// TIA Portal V17 export
// export: Created 2024-01-30T08:49:13.4989506Z, ExportSetting WithDefaults, DisplayName Totally Integrated Automation Portal, DisplayVersion V17 Update 6, DisplayName TIA Portal Openness, DisplayVersion V17 Update 6, DisplayName TIA Portal Version Control Interface, DisplayVersion V17, DisplayName STEP 7 Professional, DisplayVersion V17 Update 6, DisplayName STEP 7 Safety, DisplayVersion V17 Update 6, DisplayName WinCC Advanced, DisplayVersion V17 Update 6
FUNCTION "AnalogMeasurement" : Void   // FC2, LAD
{ S7_Optimized_Access := 'TRUE' }
VERSION : 0.1
// stored: AutoNumber true, IsIECCheckEnabled false, SetENOAutomatically false, UDAEnableTagReadback false
   VAR_INPUT
      "LK-H057_01" : Int;   // Keyence Dist.Senz-01
      "LK-H057_02" : Int;   // Keyence Dist.Senz-01
   END_VAR
   VAR_OUTPUT
      "LK-H057_01_R" : Real;
      "LK-H057_02_R" : Real;
   END_VAR
   VAR_TEMP
      Distanz_In_Prozent_01 : Real;
      Distanz_In_Prozent_02 : Real;
   END_VAR
BEGIN

REGION Network 1: LK-H057_01 Analog Werte
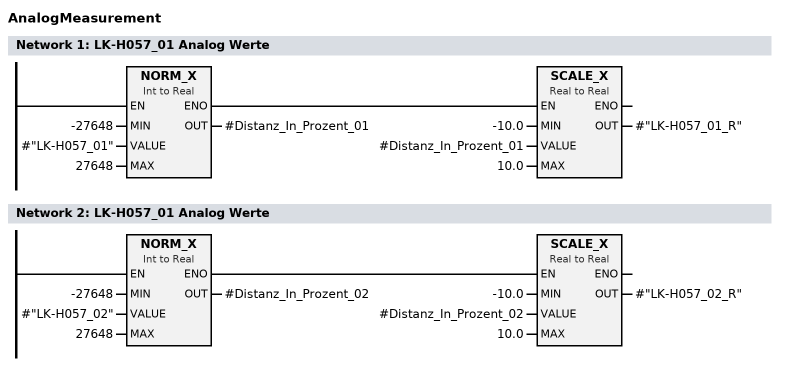
   RUNG wire#powerrail
      { S7_Templates := "[SrcType := Int, DestType := Real]" } Normalize(min := -27648, value := #"LK-H057_01", max := 27648, out => #Distanz_In_Prozent_01)
      { S7_Templates := "[SrcType := Real, DestType := Real]" } Scale(min := -10.0, value := #Distanz_In_Prozent_01, max := 10.0, out => #"LK-H057_01_R")
   END_RUNG
   // the same network as SCL:
   #Distanz_In_Prozent_01 := NORM_X(MIN := -27648, VALUE := #"LK-H057_01", MAX := 27648);
   #"LK-H057_01_R" := SCALE_X(MIN := -10.0, VALUE := #Distanz_In_Prozent_01, MAX := 10.0);
END_REGION

REGION Network 2: LK-H057_01 Analog Werte
   RUNG wire#powerrail
      { S7_Templates := "[SrcType := Int, DestType := Real]" } Normalize(min := -27648, value := #"LK-H057_02", max := 27648, out => #Distanz_In_Prozent_02)
      { S7_Templates := "[SrcType := Real, DestType := Real]" } Scale(min := -10.0, value := #Distanz_In_Prozent_02, max := 10.0, out => #"LK-H057_02_R")
   END_RUNG
   // the same network as SCL:
   #Distanz_In_Prozent_02 := NORM_X(MIN := -27648, VALUE := #"LK-H057_02", MAX := 27648);
   #"LK-H057_02_R" := SCALE_X(MIN := -10.0, VALUE := #Distanz_In_Prozent_02, MAX := 10.0);
END_REGION
END_FUNCTION
